FUNCTION_BLOCK FB_PowerSupply
VAR_INPUT
	nMaxVoltage						: UDINT;
	nMaxPower						: DINT;
	nMaxCurrent						: UINT;
	
	nCurrentFromPowerSupply			: UINT;
	nVoltageFromPowerSupply			: UINT;
	
	nReferenceVoltage				: UINT;  //Reference Voltage 
END_VAR

VAR_OUTPUT
	nVoltage						: UINT;
	nCurrent						: UINT;
	nPower							: UINT;
	bREMSB							: BOOL;
END_VAR
VAR
	nTargetVoltage					: UDINT;
	nTargetPower					: UDINT;
	nTargetCurrent					: UDINT;
END_VAR

bREMSB := TRUE;

PROPERTY CurrentCurrent : UINT
GET
CurrentCurrent := nCurrentFromPowerSupply * nMaxCurrent/nReferenceVoltage;
END_GET
END_PROPERTY

PROPERTY CurrentVoltage : UINT
GET
CurrentVoltage := UDINT_TO_UINT(nVoltageFromPowerSupply * nMaxVoltage/nReferenceVoltage);
END_GET
END_PROPERTY

{attribute 'TcRpcEnable'}
METHOD SwitchOff
nVoltage := 0;
nCurrent := 0;
nPower := 0;
END_METHOD

{attribute 'TcRpcEnable'}
METHOD SwitchOn
nVoltage := UDINT_TO_UINT(nTargetVoltage);
nCurrent := UDINT_TO_UINT(nTargetCurrent);
nPower := UDINT_TO_UINT(nTargetPower);
END_METHOD

PROPERTY TargetCurrent : UDINT
GET
TargetCurrent := nTargetCurrent * nMaxCurrent/nReferenceVoltage;
END_GET
SET
IF TargetCurrent < nMaxCurrent THEN
	nTargetCurrent := TargetCurrent * nReferenceVoltage / nMaxCurrent;
ELSE
	nTargetCurrent := 32767;
END_IF
END_SET
END_PROPERTY

PROPERTY TargetPower : UDINT
GET
TargetPower := UDINT_TO_UINT(nTargetPower * nMaxPower/nReferenceVoltage);
END_GET
SET
IF TargetPower < nMaxPower THEN
	nTargetPower := UDINT_TO_UINT(TargetPower * nReferenceVoltage / nMaxPower);
ELSE
	nTargetPower := 32767;
END_IF
END_SET
END_PROPERTY

PROPERTY TargetVoltage : UDINT
GET
TargetVoltage := nTargetVoltage * nMaxVoltage/nReferenceVoltage;
END_GET
SET
IF TargetVoltage < nMaxVoltage THEN
	nTargetVoltage := TargetVoltage * nReferenceVoltage/nMaxVoltage;	
	ADSLOGSTR(msgCtrlMask := ADSLOG_MSGTYPE_HINT, 
        	msgFmtStr   := 'Desired Voltage is lower than nMaxVoltage: %s', 
        	strArg      := UDINT_TO_STRING(TargetVoltage)
    		);  
ELSE
	nTargetVoltage := 32767;
	ADSLOGSTR(msgCtrlMask := ADSLOG_MSGTYPE_HINT, 
        	msgFmtStr   := 'Desired Voltage is higher than nMaxVoltage: %s', 
        	strArg      := UDINT_TO_STRING(TargetVoltage)
    		);  
END_IF
END_SET
END_PROPERTY

END_FUNCTION_BLOCK

(* stored: Version 1.1.0.1, ProductVersion 3.1.4024.11
   POU FB_PowerSupply: Id {694a453a-0e4c-4960-a1f7-c8c02c5c966b}, SpecialFunc None
   Property CurrentCurrent: Id {a246868a-ba71-48e9-9896-2b08ca3d4ff3}
   Get Get: Id {bf7362a7-3785-4939-b009-d47037af8596}
   Property CurrentVoltage: Id {3d9b079d-b735-4142-af37-f5b7ebda1a0c}
   Get Get: Id {d81ca134-74ae-4c2a-b41c-4cd6d60e5feb}
   Method SwitchOff: Id {406dab0c-c3e4-4232-9c80-67c79b87fe18}
   Method SwitchOn: Id {9eac384c-11d4-43b4-a0fd-342805cfe863}
   Property TargetCurrent: Id {d343f563-dc2f-4ba3-a5a7-3e8121e2a766}
   Get Get: Id {585aae2f-bc46-4e18-be91-dde0c664beb6}
   Set Set: Id {085509d1-6e2e-4b1b-8ff1-afe22a9fd03e}
   Property TargetPower: Id {1014a120-1881-45f0-b94a-9732201537b5}
   Get Get: Id {be726a65-190c-41c6-8fc1-3f96a7d85c64}
   Set Set: Id {9188b96a-589d-4b46-ba10-202af631135e}
   Property TargetVoltage: Id {7ef3f35e-3d08-494d-a6bc-ff6f23787064}
   Get Get: Id {18c39cb4-9b3c-4096-b002-e3c74cb3eb02}
   Set Set: Id {2c0b7b25-4e40-4b6c-b65f-6839ac12aeeb} *)
